PROGRAM p_Shakers
VAR
END_VAR

END_PROGRAM

(* stored: Version 1.1.0.1, ProductVersion 3.1.4022.18
   POU p_Shakers: Id {017c063a-5f09-4d50-9c5d-ffc48aeba37a}, SpecialFunc None *)
